{attribute 'GeneratedUsingTerminal: EL6201-0000-0017'}
{attribute addProperty BoxType "EL6201-0000-0017"}
{attribute addProperty Id "Slave_4A_DI0BOOL1Slave_4A_DI1BOOL1Slave_4A_DI2BOOL1Slave_4A_DI3BOOL1Slave_4B_DI0BOOL1Slave_4B_DI1BOOL1Slave_4B_DI2BOOL1Slave_4B_DI3BOOL1"}
{attribute addProperty CRC "2602663556"}
{attribute addProperty Size "8"}
TYPE Slave_4_Inputs_9B217E84 :
STRUCT
	{attribute addProperty Name "Slave_4A_DI0"}
	Slave_4A_DI0 : BOOL;
	{attribute addProperty Name "Slave_4A_DI1"}
	Slave_4A_DI1 : BOOL;
	{attribute addProperty Name "Slave_4A_DI2"}
	Slave_4A_DI2 : BOOL;
	{attribute addProperty Name "Slave_4A_DI3"}
	Slave_4A_DI3 : BOOL;
	{attribute addProperty Name "Slave_4B_DI0"}
	Slave_4B_DI0 : BOOL;
	{attribute addProperty Name "Slave_4B_DI1"}
	Slave_4B_DI1 : BOOL;
	{attribute addProperty Name "Slave_4B_DI2"}
	Slave_4B_DI2 : BOOL;
	{attribute addProperty Name "Slave_4B_DI3"}
	Slave_4B_DI3 : BOOL;
END_STRUCT
END_TYPE

(* stored: Version 1.2.0.0, ProductVersion 3.1.4024.9
   DUT Slave_4_Inputs_9B217E84: Id {fa5301b6-9c8c-4b16-89fc-e23fb9384919} *)
